{attribute 'qualified_only'}
{attribute 'strict'}
TYPE E_Buttons :
(
	enum_member := 0
);
END_TYPE

(* stored: Version 1.1.0.1, ProductVersion 3.1.4024.10
   DUT E_Buttons: Id {827b5d9c-ed34-4267-9b88-6c4561ff1f4e} *)
